PROGRAM MAIN
VAR
END_VAR

Motion01();
Test_SDO();

END_PROGRAM

(* stored: Version 1.1.0.1, ProductVersion 3.1.4024.10
   POU MAIN: Id {7375c92f-faf1-4240-9920-cc3c7379fb74}, SpecialFunc None *)
